Universal Robots PolyScope program: remote_control_V4.0.urp

Program remote_control_V4.0 (installation=remote_contol_V4.0 directory=/programs/usbdisk/new folder createdIn=3.2.19275.0 lastSavedIn=5.11.11.1010533 robotSerialNumber=20215300207)
Calibrated DH parameters: a=[-0.00004, -0.193552, -0.164677, 0.000021, -0.000085, 0]; d=[0.151949, 47.504146, 9.837748, -57.210549, 0.085444, 0.092331]; alpha=[1.570307, 0.003126, 0.002369, 1.571485, -1.572138, 0]; deltaTheta=[0, 0.654496, 0.035211, -0.689712, 0.000001, 0]
InitVariablesNode variables(variable(name=accel, expression=0), variable(name=blend_radius, expression=0), variable(name=move_type, expression=0), variable(name=speed, expression=0), variable(name=start, expression=0), variable(name=status, expression=0), variable(name=tool, expression=0))
BeforeStart
  Script: rtde_set_watchdog("input_int_register_0", 2, "PAUSE")
  Call initialize_variables
  Set NoAction tcp=OnRobot_Default
  Call sync_registers
  Wait Sleep waitTime=0.5
Robot Program (runOnlyOnce=false)
  Script: sync()
  Script: status = 1
  Wait Condition expression=start == 1
  Script: status = 2
  Switch expression=move_type
    Case (caseValue=1)
      URCap 2FG Grip (OnRobot, OnRobot A/S) dataModel(external_internal_action.index=1, twofg.internal-grip.target-width=0.02, twofg.external-grip.target-width=0.006, twofg.target-speed=64, twofg.target-force=20)
      Script: tool = 1
      Script: write_output_integer_register(1, tool)
      Script: sync()
      Wait Sleep waitTime=1
    Case (caseValue=2)
      URCap 2FG Release (OnRobot, OnRobot A/S) dataModel(external_internal_action.index=1, twofg.internal-grip.target-width=0.05, twofg.external-grip.target-width=0.036, twofg.target-speed=20)
      Script: tool = 0
      Script: write_output_integer_register(1, tool)
      Script: sync()
      Wait Sleep waitTime=1
    Case (caseValue=3)
      Popup Warning (haltProgram=false message=Warning!, movel movement with joint data could result in collisions,if isn't a mistake, you can skip this warning inputType=Text)
      If tmpl_joint != [0,0,0,0,0,0]
        Script: movel(tmpl_joint,accel,speed,0,blend_radius)
    Case (caseValue=4)
      If tmpl_cartesian != p[0,0,0,0,0,0]
        Script: movel(tmpl_cartesian,accel,speed,0,blend_radius)
    Case (caseValue=5)
      If tmpj_joint != [0,0,0,0,0,0]
        Script: movej(tmpj_joint,accel,speed,0,blend_radius)
    Case (caseValue=6)
      Popup Warning (haltProgram=false message=Warning!, movej movement with cartesian data could result in collisions,if isn't a mistake, you can skip this warning inputType=Text)
      If tmpj_cartesian != p[0,0,0,0,0,0]
        Script: movej(tmpj_cartesian,accel,speed,0,blend_radius)
    SuppressedNode
      Case (caseValue=2147483647)
        Popup Message (haltProgram=false message=no move type selected inputType=Text)
  Script: status = 3
  Wait Condition expression=start == 0
Thread Thread_1 (runOnlyOnce=false)
  setp := Joint_6_name
  Loop Forever
    Call sync_registers
SubProgram -> sync_registers
SubProgram -> initialize_variables
SubProgram initialize_variables (keepSynchronizedWithDisk=false)
  setp := Joint_6_name
  status := 0
  start := 0
  move_type := 0
  speed := 0.0
  accel := 0.0
  blend_radius := 0.0
  tool := 0
  var_1 := GP_bool_in[64]
  var_2 := GP_bool_in[65]
SubProgram sync_registers (keepSynchronizedWithDisk=false) programFile=/programs/sync_registers.urp
  Script: sync()
  'outputs'
  Script: write_output_integer_register(0, status)
  SuppressedNode
    Script: write_output_integer_register(1, tool)
  'inputs'
  Script: move_type = read_input_integer_register(20)
  Script: start = read_input_integer_register(1)
  'set targets'
  tmp := [0,0,0,0,0,0]
  Script: tmp[0] = read_input_float_register(0)
  Script: tmp[1] = read_input_float_register(1)
  Script: tmp[2] = read_input_float_register(2)
  Script: tmp[3] = read_input_float_register(3)
  Script: tmp[4] = read_input_float_register(4)
  Script: tmp[5] = read_input_float_register(5)
  tmpl_cartesian := p[tmp[0],tmp[1],tmp[2],tmp[3],tmp[4],tmp[5]]
  tmpl_joint := [tmp[0],tmp[1],tmp[2],tmp[3],tmp[4],tmp[5]]
  tmpj_cartesian := p[tmp[0],tmp[1],tmp[2],tmp[3],tmp[4],tmp[5]]
  tmpj_joint := [tmp[0],tmp[1],tmp[2],tmp[3],tmp[4],tmp[5]]
  'speed and acceleration variables'
  Script: accel = read_input_float_register(20)
  Script: speed = read_input_float_register(21)
  Script: blend_radius = read_input_float_register(22)
  var_1 := GP_bool_in[64]
  var_2 := GP_bool_in[65]
  Script: sync()
